// TIA Portal V19 export
FUNCTION_BLOCK "Peeler_FB"   // FB43, LAD
TITLE = LOWER PEELER
// stored: MemoryReserve 100, SetENOAutomatically false
   VAR_INPUT
      AreaInterface : "AreaInterface";
      ZSI : "udt_ZoneSafetyInterface";
      DSI : Struct
         LIft : "udt_DeviceSafetyInterface";
         Extension : "udt_DeviceSafetyInterface";
      END_STRUCT;
      DataIn : Struct
         Lift : "ValveMachine_DataIn";
         Extension : "ValveMachine_DataIn";
      END_STRUCT;
      CIn : Struct
         Manager : "Peeler_Manager";
         PressureRunning : Bool;
      END_STRUCT;
      Config : Struct
         Lift : "ValveMachine_Config";
         Extension : "ValveMachine_Config";
      END_STRUCT;
   END_VAR
   VAR_OUTPUT
      MachineInterface : "MachineInterface";
      DataOut : Struct
         Lift : "ValveMachine_DataOut";
         Extension : "ValveMachine_DataOut";
      END_STRUCT;
      COut : "Peeler_Status";
   END_VAR
   VAR
      Warning : Struct
         Lift { ExternalAccessible := 'False'; ExternalVisible := 'False'; ExternalWritable := 'False'} : "ValveMachine_Wng";
         Extension { ExternalAccessible := 'False'; ExternalVisible := 'False'; ExternalWritable := 'False'} : "ValveMachine_Wng";
      END_STRUCT;
      Alarm : Struct
         Lift : "ValveAlr";
         Extension : "ValveAlr";
      END_STRUCT;
      Sts : Struct
         dummy : Bool;
      END_STRUCT;
      Ctrl : Struct
         Move_Dwn_Aut : Bool;
         Move_Up_Aut : Bool;
      END_STRUCT;
      Lift : "ValveMachine_FB";
      Extension : "ValveMachine_FB";
   END_VAR
   VAR_TEMP   // added for the SCL form of the ladder/FBD networks
      _w1 : Bool;
   END_VAR
BEGIN

REGION Network 1: Aut move
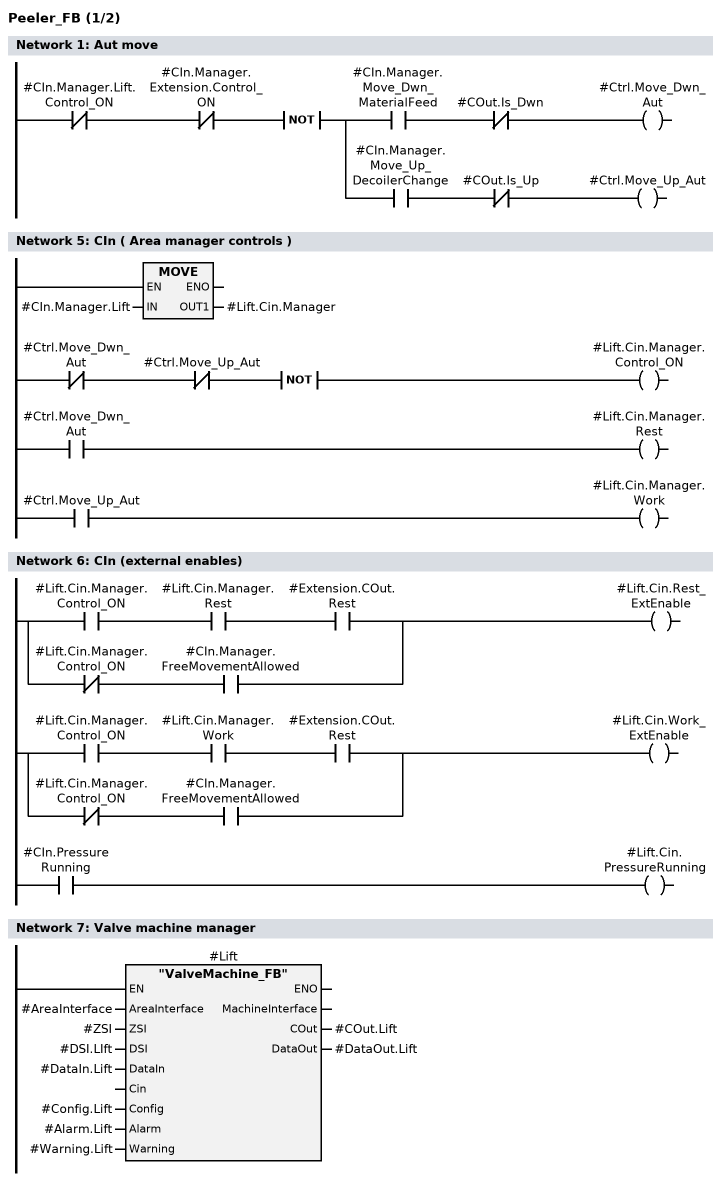
   RUNG wire#powerrail
      I_Contact( #CIn.Manager.Lift.Control_ON )
      I_Contact( #CIn.Manager.Extension.Control_ON )
      Not()
      wire#w1
      Contact( #CIn.Manager.Move_Dwn_MaterialFeed )
      I_Contact( #COut.Is_Dwn )
      Coil( #Ctrl.Move_Dwn_Aut )
   END_RUNG
   RUNG wire#w1
      Contact( #CIn.Manager.Move_Up_DecoilerChange )
      I_Contact( #COut.Is_Up )
      Coil( #Ctrl.Move_Up_Aut )
   END_RUNG
   // the same network as SCL:
   #_w1 := NOT (NOT #CIn.Manager.Lift.Control_ON AND NOT #CIn.Manager.Extension.Control_ON);
   #Ctrl.Move_Dwn_Aut := #_w1 AND #CIn.Manager.Move_Dwn_MaterialFeed AND NOT #COut.Is_Dwn;
   #Ctrl.Move_Up_Aut := #_w1 AND #CIn.Manager.Move_Up_DecoilerChange AND NOT #COut.Is_Up;
END_REGION

REGION Network 2: >
END_REGION

REGION Network 3: >
END_REGION

REGION Network 4: <<< LIFT (REST = DOWN / WORK = UP)>>>
END_REGION

REGION Network 5: CIn ( Area manager controls )
   RUNG wire#powerrail
      Move(in := #CIn.Manager.Lift, out1 => #Lift.Cin.Manager)
   END_RUNG
   RUNG wire#powerrail
      I_Contact( #Ctrl.Move_Dwn_Aut )
      I_Contact( #Ctrl.Move_Up_Aut )
      Not()
      Coil( #Lift.Cin.Manager.Control_ON )
   END_RUNG
   RUNG wire#powerrail
      Contact( #Ctrl.Move_Dwn_Aut )
      Coil( #Lift.Cin.Manager.Rest )
   END_RUNG
   RUNG wire#powerrail
      Contact( #Ctrl.Move_Up_Aut )
      Coil( #Lift.Cin.Manager.Work )
   END_RUNG
   // the same network as SCL:
   #Lift.Cin.Manager := #CIn.Manager.Lift;
   #Lift.Cin.Manager.Control_ON := NOT (NOT #Ctrl.Move_Dwn_Aut AND NOT #Ctrl.Move_Up_Aut);
   #Lift.Cin.Manager.Rest := #Ctrl.Move_Dwn_Aut;
   #Lift.Cin.Manager.Work := #Ctrl.Move_Up_Aut;
END_REGION

REGION Network 6: CIn (external enables)
   RUNG wire#powerrail
      Contact( #Lift.Cin.Manager.Control_ON )
      Contact( #Lift.Cin.Manager.Rest )
      Contact( #Extension.COut.Rest )
      wire#w1
      Coil( #Lift.Cin.Rest_ExtEnable )
   END_RUNG
   RUNG wire#powerrail
      I_Contact( #Lift.Cin.Manager.Control_ON )
      Contact( #CIn.Manager.FreeMovementAllowed )
   END_RUNG wire#w1
   RUNG wire#powerrail
      Contact( #Lift.Cin.Manager.Control_ON )
      Contact( #Lift.Cin.Manager.Work )
      Contact( #Extension.COut.Rest )
      wire#w2
      Coil( #Lift.Cin.Work_ExtEnable )
   END_RUNG
   RUNG wire#powerrail
      I_Contact( #Lift.Cin.Manager.Control_ON )
      Contact( #CIn.Manager.FreeMovementAllowed )
   END_RUNG wire#w2
   RUNG wire#powerrail
      Contact( #CIn.PressureRunning )
      Coil( #Lift.Cin.PressureRunning )
   END_RUNG
   // the same network as SCL:
   #Lift.Cin.Rest_ExtEnable := (#Lift.Cin.Manager.Control_ON AND #Lift.Cin.Manager.Rest AND #Extension.COut.Rest) OR (NOT #Lift.Cin.Manager.Control_ON AND #CIn.Manager.FreeMovementAllowed);
   #Lift.Cin.Work_ExtEnable := (#Lift.Cin.Manager.Control_ON AND #Lift.Cin.Manager.Work AND #Extension.COut.Rest) OR (NOT #Lift.Cin.Manager.Control_ON AND #CIn.Manager.FreeMovementAllowed);
   #Lift.Cin.PressureRunning := #CIn.PressureRunning;
END_REGION

REGION Network 7: Valve machine manager
   RUNG wire#powerrail
      #Lift(AreaInterface := #AreaInterface, ZSI := #ZSI, DSI := #DSI.LIft, DataIn := #DataIn.Lift, Cin :=, Config := #Config.Lift, Alarm := #Alarm.Lift, Warning := #Warning.Lift, MachineInterface =>, COut => #COut.Lift, DataOut => #DataOut.Lift)
   END_RUNG
   // the same network as SCL:
   #Lift(AreaInterface := #AreaInterface,   // "ValveMachine_FB"
         ZSI := #ZSI,
         DSI := #DSI.LIft,
         DataIn := #DataIn.Lift,
         Config := #Config.Lift,
         Alarm := #Alarm.Lift,
         Warning := #Warning.Lift,
         COut => #COut.Lift,
         DataOut => #DataOut.Lift);
END_REGION

REGION Network 8: >
END_REGION

REGION Network 9: >
END_REGION

REGION Network 10: >
END_REGION

REGION Network 11: <<< EXTENSION (REST = BKW / WORK = FWD>>>
END_REGION

REGION Network 12: CIn ( Area manager controls )
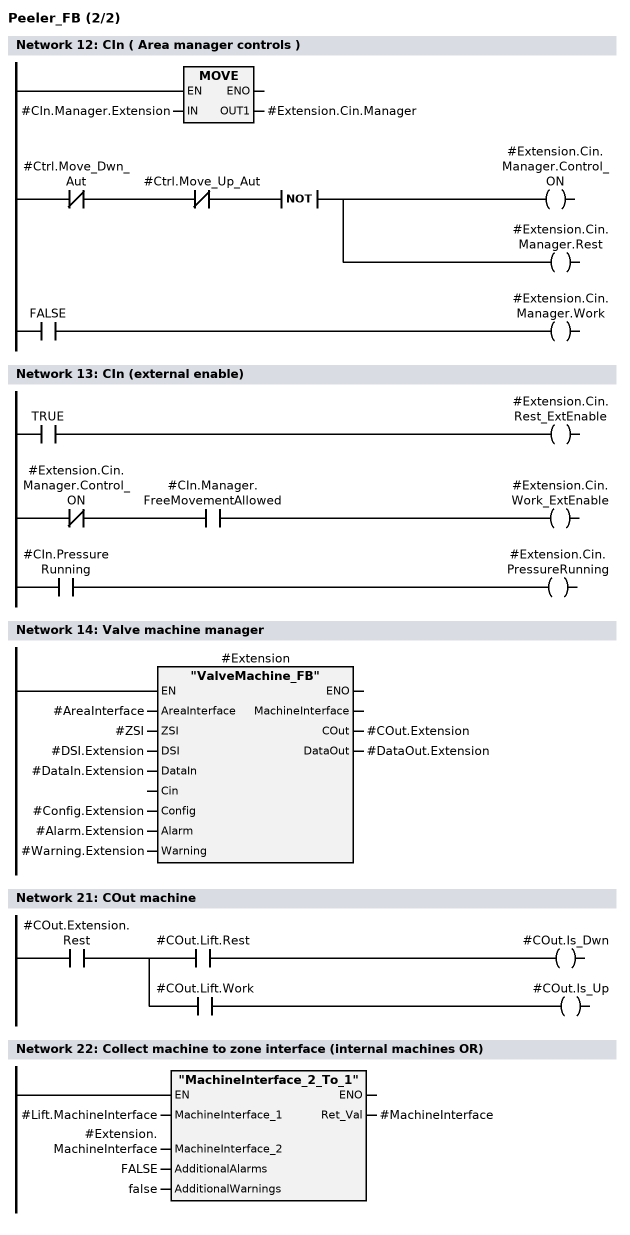
   RUNG wire#powerrail
      Move(in := #CIn.Manager.Extension, out1 => #Extension.Cin.Manager)
   END_RUNG
   RUNG wire#powerrail
      I_Contact( #Ctrl.Move_Dwn_Aut )
      I_Contact( #Ctrl.Move_Up_Aut )
      Not()
      wire#w1
      Coil( #Extension.Cin.Manager.Control_ON )
   END_RUNG
   RUNG wire#w1
      Coil( #Extension.Cin.Manager.Rest )
   END_RUNG
   RUNG wire#powerrail
      Contact( FALSE )
      Coil( #Extension.Cin.Manager.Work )
   END_RUNG
   // the same network as SCL:
   #Extension.Cin.Manager := #CIn.Manager.Extension;
   #Extension.Cin.Manager.Control_ON := NOT (NOT #Ctrl.Move_Dwn_Aut AND NOT #Ctrl.Move_Up_Aut);
   #Extension.Cin.Manager.Rest := #Extension.Cin.Manager.Control_ON;
   #Extension.Cin.Manager.Work := FALSE;
END_REGION

REGION Network 13: CIn (external enable)
   RUNG wire#powerrail
      Contact( TRUE )
      Coil( #Extension.Cin.Rest_ExtEnable )
   END_RUNG
   RUNG wire#powerrail
      I_Contact( #Extension.Cin.Manager.Control_ON )
      Contact( #CIn.Manager.FreeMovementAllowed )
      Coil( #Extension.Cin.Work_ExtEnable )
   END_RUNG
   RUNG wire#powerrail
      Contact( #CIn.PressureRunning )
      Coil( #Extension.Cin.PressureRunning )
   END_RUNG
   // the same network as SCL:
   #Extension.Cin.Rest_ExtEnable := TRUE;
   #Extension.Cin.Work_ExtEnable := NOT #Extension.Cin.Manager.Control_ON AND #CIn.Manager.FreeMovementAllowed;
   #Extension.Cin.PressureRunning := #CIn.PressureRunning;
END_REGION

REGION Network 14: Valve machine manager
   RUNG wire#powerrail
      #Extension(AreaInterface := #AreaInterface, ZSI := #ZSI, DSI := #DSI.Extension, DataIn := #DataIn.Extension, Cin :=, Config := #Config.Extension, Alarm := #Alarm.Extension, Warning := #Warning.Extension, MachineInterface =>, COut => #COut.Extension, DataOut => #DataOut.Extension)
   END_RUNG
   // the same network as SCL:
   #Extension(AreaInterface := #AreaInterface,   // "ValveMachine_FB"
              ZSI := #ZSI,
              DSI := #DSI.Extension,
              DataIn := #DataIn.Extension,
              Config := #Config.Extension,
              Alarm := #Alarm.Extension,
              Warning := #Warning.Extension,
              COut => #COut.Extension,
              DataOut => #DataOut.Extension);
END_REGION

REGION Network 15: >
END_REGION

REGION Network 16: >
END_REGION

REGION Network 17: >
END_REGION

REGION Network 18: >
END_REGION

REGION Network 19: >
END_REGION

REGION Network 20: <<< MACHINE STATUS >>>
END_REGION

REGION Network 21: COut machine
   RUNG wire#powerrail
      Contact( #COut.Extension.Rest )
      wire#w1
      Contact( #COut.Lift.Rest )
      Coil( #COut.Is_Dwn )
   END_RUNG
   RUNG wire#w1
      Contact( #COut.Lift.Work )
      Coil( #COut.Is_Up )
   END_RUNG
   // the same network as SCL:
   #COut.Is_Dwn := #COut.Extension.Rest AND #COut.Lift.Rest;
   #COut.Is_Up := #COut.Extension.Rest AND #COut.Lift.Work;
END_REGION

REGION Network 22: Collect machine to zone interface (internal machines OR)
   RUNG wire#powerrail
      "MachineInterface_2_To_1"(MachineInterface_1 := #Lift.MachineInterface, MachineInterface_2 := #Extension.MachineInterface, AdditionalAlarms := FALSE, AdditionalWarnings := false, Ret_Val => #MachineInterface)
   END_RUNG
   // the same network as SCL:
   #MachineInterface := "MachineInterface_2_To_1"(MachineInterface_1 := #Lift.MachineInterface,
                           MachineInterface_2 := #Extension.MachineInterface,
                           AdditionalAlarms := FALSE,
                           AdditionalWarnings := false);
END_REGION

REGION Network 23: >
END_REGION

REGION Network 24: >
END_REGION
END_FUNCTION_BLOCK
